// TIA Portal V16 export
// export: Created 2023-03-29T11:03:37.9694151Z, ExportSetting WithDefaults, DisplayName Totally Integrated Automation Portal, DisplayVersion V16 Update 6, DisplayName TIA Portal Version Control Interface, DisplayVersion V16 Update 2, DisplayName TIA Portal Openness, DisplayVersion V16 Update 6, DisplayName STEP 7 Professional, DisplayVersion V16 Update 6, DisplayName STEP 7 Safety, DisplayVersion V16, DisplayName WinCC Advanced, DisplayVersion V16 Update 6
DATA_BLOCK "MB_CLIENT_Send_DB"   // DB2
// stored: AutoNumber true, DBAccessibleFromOPCUA true, InstanceOfName MB_CLIENT, OfSystemLibElement MB_CLIENT, OfSystemLibVersion 3.1
"MB_CLIENT"
   // VAR_INPUT
   //    REQ : Bool;
   //    DISCONNECT : Bool;
   //    CONNECT_ID : UInt;
   //    IP_OCTET_1 : USInt;
   //    IP_OCTET_2 : USInt;
   //    IP_OCTET_3 : USInt;
   //    IP_OCTET_4 : USInt;
   //    IP_PORT : UInt;
   //    MB_MODE : USInt;
   //    MB_DATA_ADDR : UDInt;
   //    MB_DATA_LEN : UInt;
   // END_VAR
   // VAR_OUTPUT
   //    DONE : Bool;
   //    BUSY : Bool;
   //    ERROR : Bool;
   //    STATUS : Word;
   // END_VAR
   // VAR_IN_OUT
   //    MB_DATA_PTR : Variant;
   // END_VAR
   // VAR
   //    TCON_SFB { S7_SetPoint := 'True'} : TCON;
   //    TDISCON_SFB { S7_SetPoint := 'True'} : TDISCON;
   //    TSEND_SFB { S7_SetPoint := 'True'} : TSEND;
   //    TRCV_SFB { S7_SetPoint := 'True'} : TRCV;
   //    TCON_PARAM { S7_SetPoint := 'True'} : TCON_Param;
   //    PF_FREQUENCY : Real;
   //    BLOCKED_PROC_TIMEOUT : Real;
   //    RCV_TIMEOUT : Real;
   //    CURRENT_TIME_VALUE : DWord;
   //    SAVED_TIME_VALUE : DWord;
   //    XMT_TIME : DWord;
   //    SAVED_CONNECT_ID : Word;
   //    SAVED_IP_PORT : Word;
   //    SAVED_MODE : Byte;
   //    SAVED_IP1 : Byte;
   //    SAVED_IP2 : Byte;
   //    SAVED_IP3 : Byte;
   //    SAVED_IP4 : Byte;
   //    SAVED_DATA_ADDR : DWord;
   //    SAVED_DATA_LEN : Word;
   //    MB_STATE : Word;
   //    COMM_SENT_COUNT : Word;
   //    BYTE_COUNT : Word;
   //    BYTE_COUNTB : Byte;
   //    SAVED_START_ADDR : Word;
   //    MB_TRANSACTION_ID : Word;
   //    MB_UNIT_ID : Word;
   //    RETRIES : Word;
   //    INIT_OK : Bool;
   //    ACTIVE : Bool;
   //    CONNECTED : Bool;
   //    SAVED_MA_REQ : Bool;
   // END_VAR
BEGIN
END_DATA_BLOCK
